(* CoDeSys 2.3 export: FB_DECODE_FEF2.EXP *)

(* POU PGN FB/FB_DECODE_FEF2, ST *)
FUNCTION_BLOCK FB_DECODE_FEF2
VAR_IN_OUT
	IN: ARRAY [0..7] OF USINT;
END_VAR
VAR_OUTPUT
	EngineFuelRate : REAL;

	Count : DWORD;
END_VAR
VAR
	Debug : BOOL;
	Buffer: ARRAY [0..7] OF USINT;
END_VAR
EngineFuelRate := BUFFER_TO_REAL( pBuffer:= ADR(IN[0]), ByteSize := 2, Scale:= 0.05, Offset := 0.0 );

Count := Count + 1;

IF Debug THEN MEMCPY(destAddr := ADR(Buffer), srcAddr := ADR(IN), n := 8); END_IF
END_FUNCTION_BLOCK
